{attribute addProperty BoxType "EL3423-0000-0016"}
{attribute addProperty Id "PQF_AvgAT %I*REAL32417PQF_MinAT %I*REAL32418PQF_MaxAT %I*REAL32419"}
{attribute addProperty CRC "1331830692"}
{attribute addProperty SizeInBites "96"}
{attribute addProperty SizeInBytes "12"}
TYPE Total_Statistic_PQF_4F621FA4 :
STRUCT
	{attribute addProperty Name "PQF_Avg"}
	PQF_Avg AT %I* : REAL;
	{attribute addProperty Name "PQF_Min"}
	PQF_Min AT %I* : REAL;
	{attribute addProperty Name "PQF_Max"}
	PQF_Max AT %I* : REAL;
END_STRUCT
END_TYPE

(* stored: Version 1.2.0.0, ProductVersion 3.1.4024.9
   DUT Total_Statistic_PQF_4F621FA4: Id {9e1ecd82-9253-44af-bfc9-7d5faa26a051} *)
